FUNCTION_BLOCK SufficientFeedFlow (* Extracted Composite Function Block Type *)
  (* Standard: 61499-2 *)
  (* Version 9/23/2026 *)
  PACKAGE SE.Nereda;
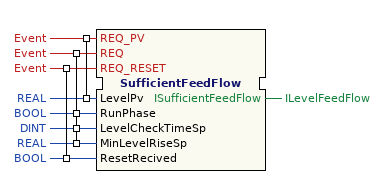
  EVENT_INPUT
    REQ_PV WITH LevelPv;
    REQ WITH RunPhase, LevelCheckTimeSp, MinLevelRiseSp; (* Normal Execution Request *)
    REQ_RESET WITH ResetRecived;
  END_EVENT
  VAR_INPUT
    LevelPv : REAL;
    RunPhase : BOOL;
    LevelCheckTimeSp : DINT;
    MinLevelRiseSp : REAL;
    ResetRecived : BOOL;
  END_VAR
  PLUGS
    ISufficientFeedFlow : ILevelFeedFlow;
  END_PLUGS
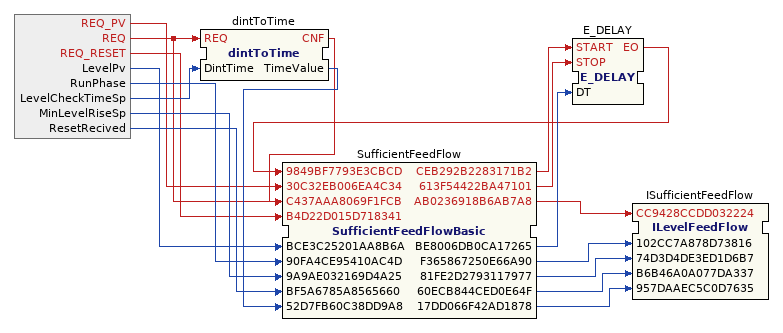
  FBS
    SufficientFeedFlow : SufficientFeedFlowBasic;
    E_DELAY : E_DELAY;
    dintToTime : dintToTime;
  END_FBS
  EVENT_CONNECTIONS
    SufficientFeedFlow.CEB292B2283171B2 TO E_DELAY.START;
    SufficientFeedFlow.613F54422BA47101 TO E_DELAY.STOP;
    E_DELAY.EO TO SufficientFeedFlow.9849BF7793E3CBCD;
    REQ_PV TO SufficientFeedFlow.30C32EB006EA4C34;
    REQ TO SufficientFeedFlow.C437AAA8069F1FCB;
    REQ_RESET TO SufficientFeedFlow.B4D22D015D718341;
    dintToTime.CNF TO SufficientFeedFlow.C437AAA8069F1FCB;
    REQ TO dintToTime.REQ;
    SufficientFeedFlow.AB0236918B6AB7A8 TO ISufficientFeedFlow.CC9428CCDD032224;
  END_CONNECTIONS
  DATA_CONNECTIONS
    LevelPv TO SufficientFeedFlow.BCE3C25201AA8B6A;
    RunPhase TO SufficientFeedFlow.90FA4CE95410AC4D;
    LevelCheckTimeSp TO dintToTime.DintTime;
    MinLevelRiseSp TO SufficientFeedFlow.9A9AE032169D4A25;
    ResetRecived TO SufficientFeedFlow.BF5A6785A8565660;
    dintToTime.TimeValue TO SufficientFeedFlow.52D7FB60C38DD9A8;
    SufficientFeedFlow.BE8006DB0CA17265 TO E_DELAY.DT;
    SufficientFeedFlow.F365867250E66A90 TO ISufficientFeedFlow.102CC7A878D73816;
    SufficientFeedFlow.81FE2D2793117977 TO ISufficientFeedFlow.74D3D4DE3ED1D6B7;
    SufficientFeedFlow.60ECB844CED0E64F TO ISufficientFeedFlow.B6B46A0A077DA337;
    SufficientFeedFlow.17DD066F42AD1878 TO ISufficientFeedFlow.957DAAEC5C0D7635;
  END_CONNECTIONS
END_FUNCTION_BLOCK
